TYPE
    InfoData :
    STRUCT
        State         : UINT; // 0 valid
        AdsAddr       : AMSADDR;
        DcOutputShift : DINT;
        DcInputShift  : DINT;
    END_STRUCT
END_TYPE

(* stored: Version 1.1.0.1, ProductVersion 3.1.4024.12
   DUT InfoData: Id {10076343-6c3a-4156-9f95-7ec64bec87d4} *)
